// Mitsubishi GX Works2 project: Class3_디바이스버퍼&Pulse   PLC: Q03UD

PROGRAM MAIN
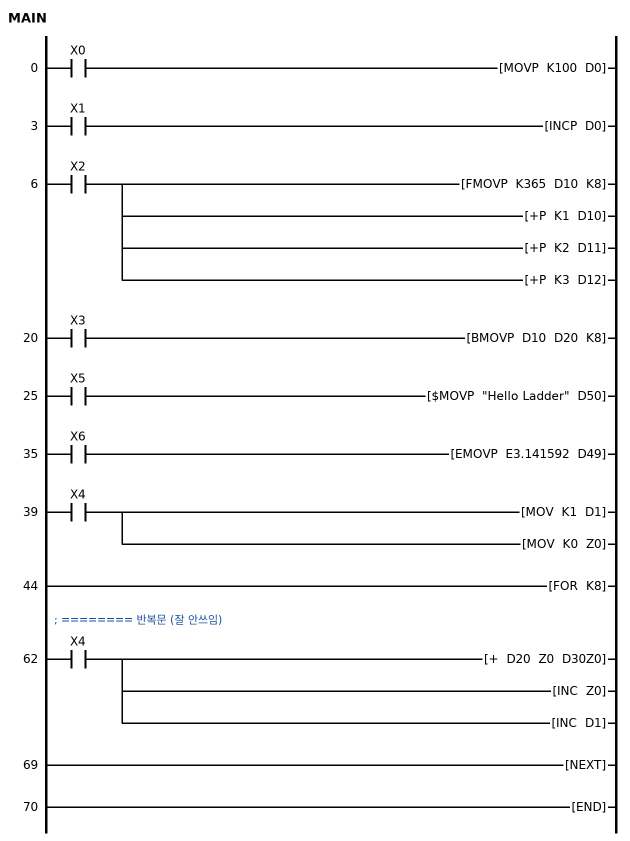
0     LD      X0
      MOVP    K100 D0
3     LD      X1
      INCP    D0
6     LD      X2
      FMOVP   K365 D10 K8
      +P      K1 D10
      +P      K2 D11
      +P      K3 D12
20    LD      X3
      BMOVP   D10 D20 K8
25    LD      X5
      $MOVP   "Hello Ladder" D50
35    LD      X6
      EMOVP   E3.141592 D49
39    LD      X4
      MOV     K1 D1
      MOV     K0 Z0
44    FOR     K8
; ======== 반복문 (잘 안쓰임)
62    LD      X4
      +       D20 Z0 D30Z0
      INC     Z0
      INC     D1
69    NEXT
70    END
END_PROGRAM
